FUNCTION_BLOCK LocalizedText2LocalizedText (* Function Block to set a connection to the LocalizedText type *)
  (* Standard: 61499-2 *)
  (* Version 1.0, 2019-07-08, TS, fortiss GmbH *)
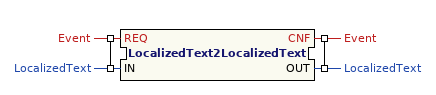
  EVENT_INPUT
    REQ WITH IN; (* Normal Execution Request *)
  END_EVENT
  EVENT_OUTPUT
    CNF WITH OUT; (* Execution Confirmation *)
  END_EVENT
  VAR_INPUT
    IN : LocalizedText; (* Input event qualifier *)
  END_VAR
  VAR_OUTPUT
    OUT : LocalizedText; (* Output event qualifier *)
  END_VAR
  (* Service APPLICATION/RESOURCE: Helper FB to set the connection to the LocalizedText type *)
END_FUNCTION_BLOCK
